TYPE TcoOmnicore_Outputs_v_1_x_x :
STRUCT
	Outputs AT %Q* : ARRAY[0..63] OF BYTE;
END_STRUCT
END_TYPE

(* stored: Version 1.1.0.1, ProductVersion 3.1.4024.12
   DUT TcoOmnicore_Outputs_v_1_x_x: Id {b739efad-2cc0-05cb-26b8-444c06eeeeb2} *)
